{attribute 'GeneratedUsingTerminal: EL7031-0030-0016'}
{attribute addProperty BoxType "EL7031-0030-0016"}
{attribute addProperty Id "AdsAddrAT %I*AMSADDR8Chn0AT %I*USINT1Chn1AT %I*USINT1Chn2AT %I*USINT1Chn3AT %I*USINT1StateAT %I*UINT2"}
{attribute addProperty CRC "2476700086"}
{attribute addProperty Size "14"}
TYPE InfoData_939F71B6 :
STRUCT
	{attribute addProperty Name "AdsAddr"}
	AdsAddr AT %I* : AMSADDR;
	{attribute addProperty Name "Chn0"}
	Chn0 AT %I* : USINT;
	{attribute addProperty Name "Chn1"}
	Chn1 AT %I* : USINT;
	{attribute addProperty Name "Chn2"}
	Chn2 AT %I* : USINT;
	{attribute addProperty Name "Chn3"}
	Chn3 AT %I* : USINT;
	{attribute addProperty Name "State"}
	State AT %I* : UINT;
END_STRUCT
END_TYPE

(* stored: Version 1.2.0.0, ProductVersion 3.1.4024.9
   DUT InfoData_939F71B6: Id {9be010ba-8990-48d5-9d17-201aace45a15} *)
